{attribute 'GeneratedUsingTerminal: EL5151-0021-0018'}
{attribute addProperty BoxType "EL5151-0021-0018"}
{attribute addProperty Id "ControlAT %Q*Control_135F4E528Set_counter_valueAT %Q*UDINT4Switch_on_threshold_valueAT %Q*UDINT4Switch_off_threshold_valueAT %Q*UDINT4"}
{attribute addProperty CRC "3949351489"}
{attribute addProperty Size "20"}
TYPE ENC_Control_EB665241 EXTENDS OutputBase_10CEE7DE :
STRUCT
	{attribute addProperty Name "Control"}
	Control AT %Q* : Control_135F4E52;
	{attribute addProperty Name "Set_counter_value"}
	Set_counter_value AT %Q* : UDINT;
	{attribute addProperty Name "Switch_on_threshold_value"}
	Switch_on_threshold_value AT %Q* : UDINT;
	{attribute addProperty Name "Switch_off_threshold_value"}
	Switch_off_threshold_value AT %Q* : UDINT;
END_STRUCT
END_TYPE

(* stored: Version 1.2.0.0, ProductVersion 3.1.4024.9
   DUT ENC_Control_EB665241: Id {12249645-f782-4bf2-b6a9-2166f19a906d} *)
